SUBAPPLICATION Uebung_234_AX (* Zweipunktregler (Fuellstand/Thermostat-Muster) via DualHysteresis_AR_A2X + A2X_TO_QXA2 - reiner Hardware-Aufbau ohne VT *)
  (* Standard: 61499-2; Description: Copyright (c) 2026 Meisterschulen am Ostbahnhof This program and the accompanying materials are made available under the terms of the Eclipse Public License 2.0 which is available at https://www.eclipse.org/legal/epl-2.0/ SPDX-License-Identifier: EPL-2.0 *)
  (* Version 1.0, 2026-09-07, Franz Höpfinger, Meisterschulen am Ostbahnhof, initial API and implementation and/or initial documentation *)
  PACKAGE Uebungen;
  IMPORT logiBUS::io::AI::logiBUS_AI::AnalogInput_I4;
  IMPORT logiBUS::io::DQ::logiBUS_DO::Output_Q1;
  IMPORT logiBUS::io::DQ::logiBUS_DO::Output_Q2;
  (* Documentation:
  Zweipunktregler mit Hysterese (reine Hardware-Übung, ohne VT)
   Klassisches Thermostat-/Füllstandsschalter-Muster: ein analoger Messwert (z.B. Füllstand oder Temperatur) wird gegen einen Mittelwert MI mit Totzone (DEAD) und Hysterese (HYSTERESIS) geprüft und steuert darüber zwei entgegengesetzte Aktoren (z.B. Befüllen/Entleeren oder Heizen/Kühlen) - nie beide gleichzeitig.
   Funktionsbeschreibung
    - AnalogInput_I4 (logiBUS_AI_IDA) liefert den rohen AD-Messwert; AD_TO_AUDI → AUDI_TO_AR wandeln ihn in eine AR (REAL-Adapter) um - dieselbe doppelte Konvertierung wie in Uebung_028a_AR ("ein AD_TO_AR wäre wie ein reinterpret_cast").
   - DualHysteresis_AR_A2X vergleicht den Messwert gegen MI (hier fest 500.0 über HysteresisParams_AR, im echten Einsatz parametrierbar): steigt der Wert über MI + DEAD + HYSTERESIS, schaltet UP ein; fällt er unter MI - DEAD - HYSTERESIS, schaltet DOWN ein. Ausgeschaltet wird erst wieder, wenn der Wert in die reine Totzone MI ± DEAD zurückkehrt - die Differenz zwischen Ein- und Ausschaltpunkt (HYSTERESIS) verhindert Flattern nahe der Schaltschwelle.
   - A2X_TO_QXA2 entbündelt das eine A2X-Ausgangssignal (UP/DOWN) auf zwei physische logiBUS-Ausgänge - siehe Doku dieses Bausteins für das "SUB style"-Prinzip dahinter.
    Arbeitsauftrag
   Testen Sie mit einem Potentiometer oder simuliertem Analogwert an AnalogInput_I4: Wert weit über 500 → Q1 (UP) EIN, Q2 (DOWN) AUS. Wert weit unter 500 → umgekehrt. Wert nahe 500 (innerhalb ±20) → beide AUS. Beobachten Sie das Hysterese-Verhalten: der Ausschaltpunkt liegt näher an MI als der Einschaltpunkt.
   Für dieselbe Funktion mit VT-Anzeige (Messwert als Zahlenfeld, UP/DOWN als Lampen) siehe Uebung_235_AX.
  *)
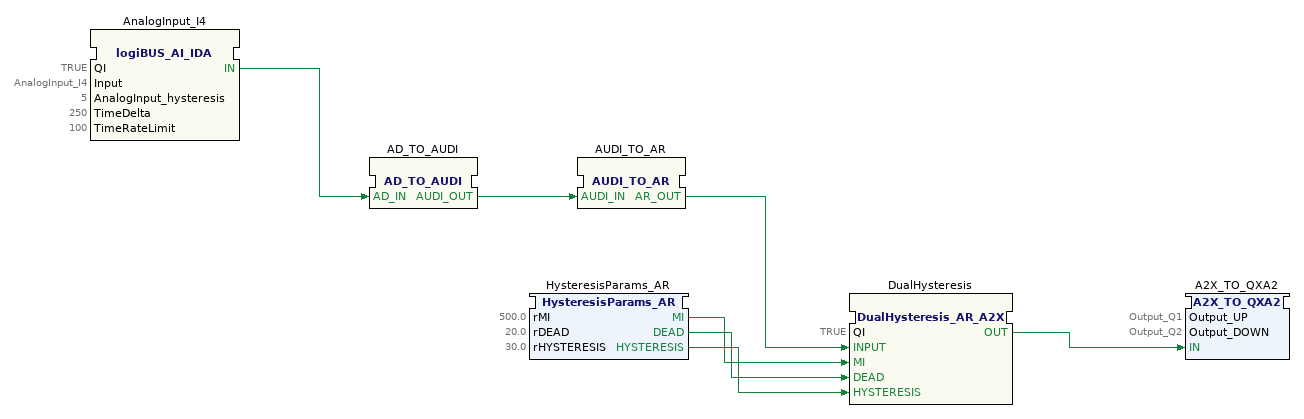
  (* Zweipunktregelung mit Totzone + Hysterese um einen Mittelwert MI: - ueber MI+DEAD+HYSTERESIS schaltet UP ein (z.B. Heizen/Befuellen), unter MI-DEAD-HYSTERESIS schaltet DOWN ein (z.B. Kuehlen/Entleeren). - Ausschalten erst innerhalb der reinen Totzone (MI +/- DEAD) - die Hysterese verhindert Flattern nahe der Schaltschwelle. - MI/DEAD/HYSTERESIS hier als feste Beispielwerte (initval_AR) - in echten Anlagen typischerweise per INI/OPC-UA parametrierbar. *)
  FBS
    AnalogInput_I4 : logiBUS::io::AI::logiBUS_AI_IDA(QI := TRUE, Input := AnalogInput_I4, AnalogInput_hysteresis := 5, TimeDelta := 250, TimeRateLimit := 100);
    AD_TO_AUDI : adapter::conversion::unidirectional::AD_TO_AUDI;
    AUDI_TO_AR : adapter::conversion::unidirectional::AUDI_TO_AR;
    DualHysteresis : logiBUS::signalprocessing::hysteresis::DualHysteresis_AR_A2X(QI := TRUE);
  END_FBS
  SUBAPPS
    HysteresisParams_AR : MyLib::sys::HysteresisParams_AR(rMI := 500.0, rDEAD := 20.0, rHYSTERESIS := 30.0);
    A2X_TO_QXA2 : MyLib::sys::A2X_TO_QXA2(Output_UP := Output_Q1, Output_DOWN := Output_Q2);
  END_SUBAPPS
  ADAPTER_CONNECTIONS
    AnalogInput_I4.IN TO AD_TO_AUDI.AD_IN;
    AD_TO_AUDI.AUDI_OUT TO AUDI_TO_AR.AUDI_IN;
    AUDI_TO_AR.AR_OUT TO DualHysteresis.INPUT;
    HysteresisParams_AR.MI TO DualHysteresis.MI;
    HysteresisParams_AR.DEAD TO DualHysteresis.DEAD;
    HysteresisParams_AR.HYSTERESIS TO DualHysteresis.HYSTERESIS;
    DualHysteresis.OUT TO A2X_TO_QXA2.IN;
  END_CONNECTIONS
END_SUBAPPLICATION
